FUNCTION_BLOCK ATV_Schneider (* Extracted Composite Function Block Type *)
  (* Standard: 61499-2 *)
  (* Version 24/02/2026 *)
  PACKAGE Hidryco.HidrycoLib;
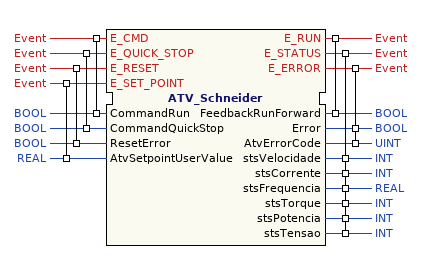
  EVENT_INPUT
    E_CMD WITH CommandRun;
    E_QUICK_STOP WITH CommandQuickStop; (* Data write request *)
    E_RESET WITH ResetError;
    E_SET_POINT WITH AtvSetpointUserValue;
  END_EVENT
  EVENT_OUTPUT
    E_RUN WITH FeedbackRunForward; (* Confirmation of an explicit or implicit data read request *)
    E_STATUS WITH stsVelocidade, stsCorrente, stsFrequencia, stsTorque, stsPotencia, stsTensao; (* Execution Confirmation *)
    E_ERROR WITH Error, AtvErrorCode;
  END_EVENT
  VAR_INPUT
    CommandRun : BOOL;
    CommandQuickStop : BOOL; (* New value(i) for the named variable element *)
    ResetError : BOOL; (* New value(i) for the named variable element *)
    AtvSetpointUserValue : REAL; (* Input in RPM for Speed Control HW CAT, Input in Hz for Frequency Control HW CAT *)
  END_VAR
  VAR_OUTPUT
    FeedbackRunForward : BOOL; (* Current value(i) in the named variable array element *)
    Error : BOOL; (* Current value(i) in the named variable array element *)
    AtvErrorCode : UINT; (* Current value(i) in the named variable array element *)
    stsVelocidade : INT; (* Result *)
    stsCorrente : INT; (* Result *)
    stsFrequencia : REAL; (* Result *)
    stsTorque : INT; (* Result *)
    stsPotencia : INT; (* Result *)
    stsTensao : INT; (* Result *)
  END_VAR
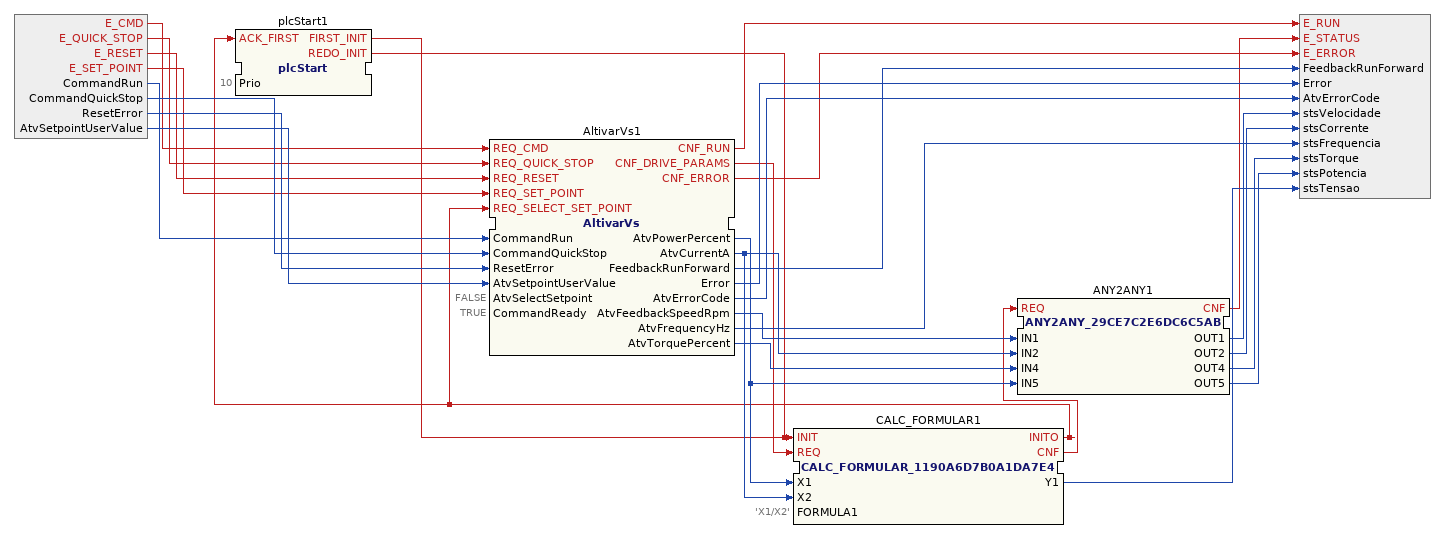
  FBS
    AltivarVs1 : AltivarVs(AtvSelectSetpoint := FALSE, CommandReady := TRUE);
    ANY2ANY1 : ANY2ANY_29CE7C2E6DC6C5AB; {SET_ATTRIBUTE(Configuration.GenericFBType.InterfaceParams, Runtime.Standard#CNT:=5;IN${CNT$}:REAL,REAL,REAL,REAL,REAL;OUT${CNT$}:INT,INT,REAL,INT,INT)}
    CALC_FORMULAR1 : CALC_FORMULAR_1190A6D7B0A1DA7E4(FORMULA1 := 'X1/X2'); {SET_ATTRIBUTE(Configuration.GenericFBType.InterfaceParams, Runtime.Standard#OUTCNT:=1;INCNT:=2;X${INCNT$}:LREAL,LREAL;Y${OUTCNT$}:INT)}
    plcStart1 : plcStart(Prio := 10);
  END_FBS
  EVENT_CONNECTIONS
    E_CMD TO AltivarVs1.REQ_CMD;
    E_QUICK_STOP TO AltivarVs1.REQ_QUICK_STOP;
    E_RESET TO AltivarVs1.REQ_RESET;
    E_SET_POINT TO AltivarVs1.REQ_SET_POINT;
    AltivarVs1.CNF_RUN TO E_RUN;
    plcStart1.FIRST_INIT TO CALC_FORMULAR1.INIT;
    plcStart1.REDO_INIT TO CALC_FORMULAR1.INIT;
    CALC_FORMULAR1.INITO TO AltivarVs1.REQ_SELECT_SET_POINT;
    CALC_FORMULAR1.INITO TO plcStart1.ACK_FIRST;
    AltivarVs1.CNF_DRIVE_PARAMS TO CALC_FORMULAR1.REQ;
    AltivarVs1.CNF_ERROR TO E_ERROR;
    CALC_FORMULAR1.CNF TO ANY2ANY1.REQ;
    ANY2ANY1.CNF TO E_STATUS;
  END_CONNECTIONS
  DATA_CONNECTIONS
    AltivarVs1.AtvPowerPercent TO CALC_FORMULAR1.X1;
    AltivarVs1.AtvCurrentA TO CALC_FORMULAR1.X2;
    CommandRun TO AltivarVs1.CommandRun;
    CommandQuickStop TO AltivarVs1.CommandQuickStop;
    ResetError TO AltivarVs1.ResetError;
    AtvSetpointUserValue TO AltivarVs1.AtvSetpointUserValue;
    AltivarVs1.FeedbackRunForward TO FeedbackRunForward;
    AltivarVs1.Error TO Error;
    AltivarVs1.AtvErrorCode TO AtvErrorCode;
    CALC_FORMULAR1.Y1 TO stsTensao;
    AltivarVs1.AtvFeedbackSpeedRpm TO ANY2ANY1.IN1;
    AltivarVs1.AtvCurrentA TO ANY2ANY1.IN2;
    AltivarVs1.AtvFrequencyHz TO stsFrequencia;
    AltivarVs1.AtvTorquePercent TO ANY2ANY1.IN4;
    AltivarVs1.AtvPowerPercent TO ANY2ANY1.IN5;
    ANY2ANY1.OUT1 TO stsVelocidade;
    ANY2ANY1.OUT2 TO stsCorrente;
    ANY2ANY1.OUT4 TO stsTorque;
    ANY2ANY1.OUT5 TO stsPotencia;
  END_CONNECTIONS
END_FUNCTION_BLOCK
